SUBAPPLICATION Uebung_010f4 (* SCHLECHTER STIL (Punktabzug!): SoftKey_F1 ODER AuxFunction2_X1 auf DigitalOutput_Q1 mit 2x GreenWhiteBackground statt GreenWhiteBackground3 - siehe Uebung_010f3 fuer die korrekte Loesung *)
  (* Standard: 61499-2; Description: Copyright (c) 2026 Meisterschulen am Ostbahnhof This program and the accompanying materials are made available under the terms of the Eclipse Public License 2.0 which is available at https://www.eclipse.org/legal/epl-2.0/ SPDX-License-Identifier: EPL-2.0 *)
  (* Version 1.0, 2026-09-06, Franz Höpfinger, Meisterschulen am Ostbahnhof, initial API and implementation and/or initial documentation *)
  PACKAGE Uebungen;
  IMPORT Uebungen::const::UT::DefaultPool::SoftKey_F1;
  IMPORT Uebungen::const::UT::DefaultPool::AuxFunction2_X1;
  IMPORT logiBUS::io::DQ::logiBUS_DO::Output_Q1;
  (* Documentation:
  SCHLECHTER STIL (Punktabzug!) - siehe Uebung_010f3 für die korrekte Lösung
   Diese Datei ist absichtlich als Negativbeispiel stehen gelassen: sie erreicht funktional dasselbe wie Uebung_010f3, tut es aber mit unnötig aufgeblähter Verdrahtung.
   Was hier falsch gemacht wurde
    - Statt des dafür gebauten Bausteins GreenWhiteBackground3 (nimmt u16ObjId UND u16ObjIdA gleichzeitig und braucht nur einen DI1-Eingang) wurden hier GreenWhiteBackground1 und GreenWhiteBackground2 als zwei separate Instanzen verdrahtet.
   - Die Farbauswahl-Logik (Weiß/Grün) läuft dadurch doppelt statt einmal - unnötiger Ressourcenverbrauch und unnötig große Diagramme, ohne jeden funktionalen Vorteil.
    Lernziel
   Bevor man für einen kombinierten Fall (normales VT-Objekt + Aux-Objekt) mehrere generische Bausteine einzeln zusammenschraubt, erst prüfen, ob es dafür nicht schon einen passenden, fertigen Baustein in der Bibliothek gibt (hier: GreenWhiteBackground3). Vergleichen Sie diese Datei mit Uebung_010f3, um den Unterschied zu sehen.
  *)
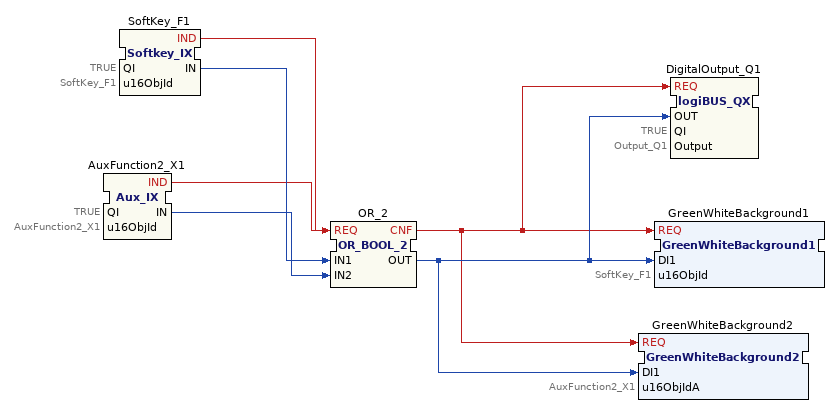
  (* SCHLECHTER STIL - Punktabzug! Hier wurden GreenWhiteBackground1 UND GreenWhiteBackground2 einzeln verdrahtet, obwohl es mit GreenWhiteBackground3 (ein Baustein, u16ObjId + u16ObjIdA) genau fuer diesen Fall (1 normales VT-Objekt + 1 Aux-Objekt) schon fertig existiert. Unnoetige Verdopplung der Farbauswahl-Logik. Korrekte Loesung: Uebung_010f3. *)
  FBS
    DigitalOutput_Q1 : logiBUS::io::DQ::logiBUS_QX(QI := TRUE, Output := Output_Q1);
    SoftKey_F1 : isobus::UT::io::Softkey::Softkey_IX(QI := TRUE, u16ObjId := SoftKey_F1);
    AuxFunction2_X1 : isobus::UT::io::Auxiliary::IN::Aux_IX(QI := TRUE, u16ObjId := AuxFunction2_X1);
    OR_2 : iec61131::booleanOperators::OR_BOOL_2;
  END_FBS
  SUBAPPS
    GreenWhiteBackground1 : MyLib::sys::GreenWhiteBackground1(u16ObjId := SoftKey_F1);
    GreenWhiteBackground2 : MyLib::sys::GreenWhiteBackground2(u16ObjIdA := AuxFunction2_X1);
  END_SUBAPPS
  EVENT_CONNECTIONS
    SoftKey_F1.IND TO OR_2.REQ;
    AuxFunction2_X1.IND TO OR_2.REQ;
    OR_2.CNF TO DigitalOutput_Q1.REQ;
    OR_2.CNF TO GreenWhiteBackground1.REQ;
    OR_2.CNF TO GreenWhiteBackground2.REQ;
  END_CONNECTIONS
  DATA_CONNECTIONS
    SoftKey_F1.IN TO OR_2.IN1;
    AuxFunction2_X1.IN TO OR_2.IN2;
    OR_2.OUT TO DigitalOutput_Q1.OUT;
    OR_2.OUT TO GreenWhiteBackground1.DI1;
    OR_2.OUT TO GreenWhiteBackground2.DI1;
  END_CONNECTIONS
END_SUBAPPLICATION
